(* PLC project Thermostats, Actility iec61131 1.0.231, author Laurent Nicq *)
(* stored: creationDateTime 2013-04-23T20:30:50, version V1.0.0, modificationDateTime 2013-07-22T15:08:27 *)

FUNCTION_BLOCK Heating_TH_PWM
  VAR_INPUT
    PWM2_Start : BOOL;
    PWM2_Period : TIME;
  END_VAR
  VAR
    PWM2_Running_ON_Time : TIME;
    PWM2_Ratio : DINT;
    PWM2_Limit_Low : DINT := 0;
  END_VAR
  VAR_INPUT
    PWM2_Limit_High : DINT;  (* If not set as INPUT, put 100.0 as initial value *)
  END_VAR
  VAR
    PWM_Ratio_Factor : DINT := 100;
    PWM2_ResetMode : DINT := 0;  (* For simulation *)
    PWM_Time_ON : TIME;
  END_VAR
  VAR_OUTPUT
    PWM2_Out : BOOL;
  END_VAR
  VAR_INPUT
    Setpoint : REAL;
    Temperature_Inside : REAL;
    Proportional_Inside : REAL;
    Temperature_Outside : REAL;
    Proportional_Outside : REAL;
  END_VAR
  VAR
    Inside_Demand : REAL;
    Outside_Demand : REAL;
    Demand_Factor : REAL := 100.0;
    PWM_HEATING : PWM_GENERATOR;
  END_VAR
  VAR  (* added by the conversion: wires and edge detectors of the diagram *)
    _SUB32_OUT : REAL;
    _MUL31_OUT : REAL;
    _SUB2_OUT : REAL;
    _MUL1_OUT : REAL;
    _ADD37_OUT : REAL;
    _MUL38_OUT : REAL;
    _REAL_TO_DINT41_OUT : DINT;
  END_VAR

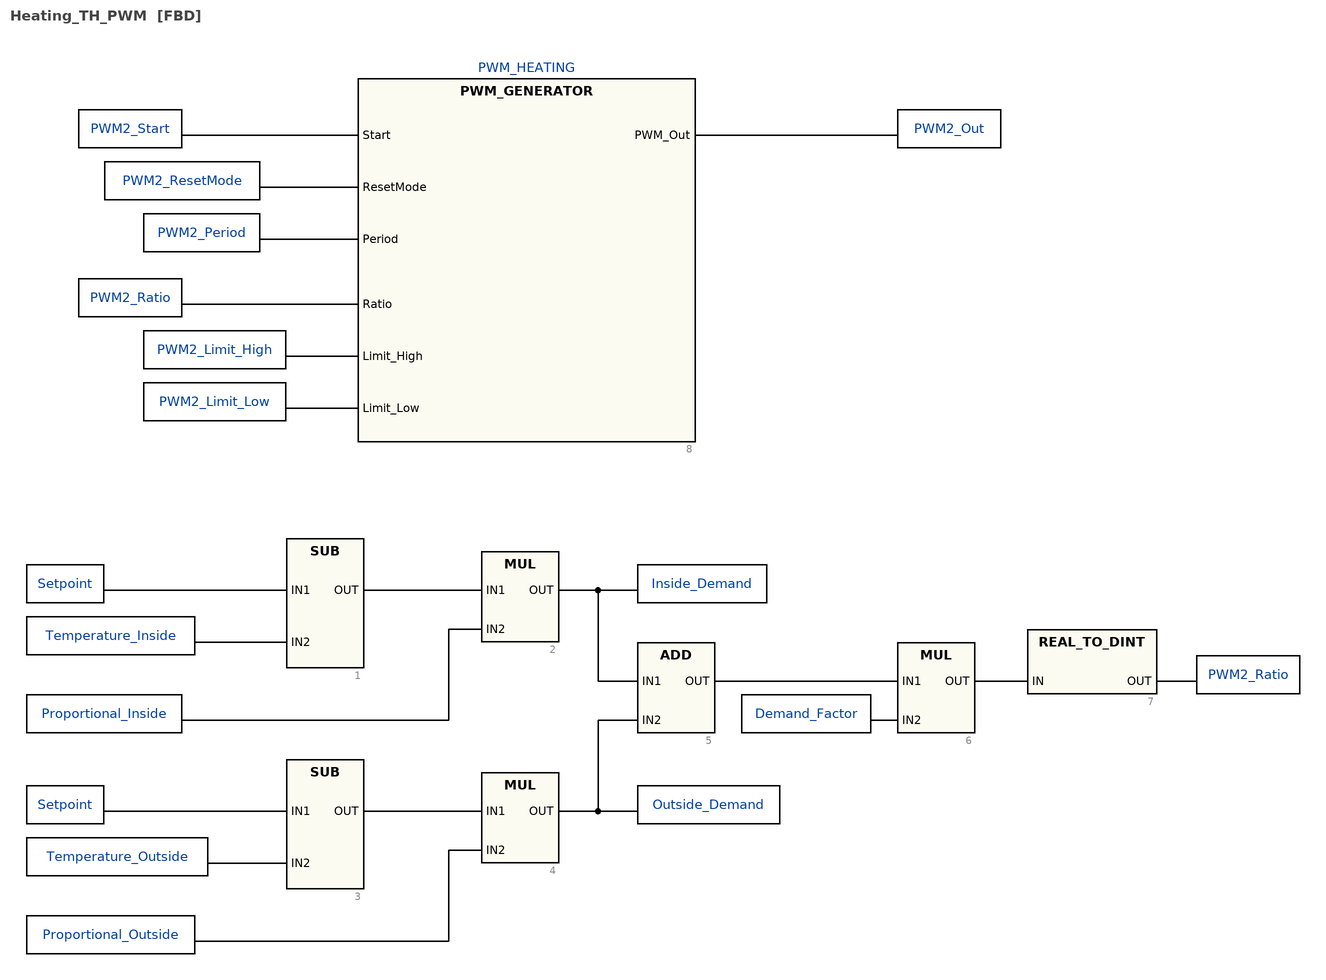
(* FBD diagram, written out as Structured Text *)
_SUB32_OUT := Setpoint - Temperature_Inside;
_MUL31_OUT := _SUB32_OUT * Proportional_Inside;
_SUB2_OUT := Setpoint - Temperature_Outside;
_MUL1_OUT := _SUB2_OUT * Proportional_Outside;
_ADD37_OUT := _MUL31_OUT + _MUL1_OUT;
_MUL38_OUT := _ADD37_OUT * Demand_Factor;
_REAL_TO_DINT41_OUT := REAL_TO_DINT(_MUL38_OUT);
PWM_HEATING(Start := PWM2_Start, ResetMode := PWM2_ResetMode, Period := PWM2_Period, Ratio := PWM2_Ratio, Limit_High := PWM2_Limit_High, Limit_Low := PWM2_Limit_Low);
PWM2_Out := PWM_HEATING.PWM_Out;
Inside_Demand := _MUL31_OUT;
PWM2_Ratio := _REAL_TO_DINT41_OUT;
Outside_Demand := _MUL1_OUT;
END_FUNCTION_BLOCK

PROGRAM Thermostat_PWM_DINT
  VAR
    TH_Period : TIME := T#20s;  (* Period in Second *)
    TH_PWM_Start : BOOL := FALSE;  (* Needs RISING Edge to start *)
    TH_Ratio_Limit_High : DINT := 100;  (* Ratio Limit High in % *)
    TH_Setpoint : REAL := 28.0;
  END_VAR
  VAR_EXTERNAL
    TH_Temp_Inside : REAL;
  END_VAR
  VAR
    TH_Temp_Outside : REAL := 12.0;
    TH_PROP_Inside : REAL := 0.5;
    TH_PROP_Outside : REAL := 0.0;
  END_VAR
  VAR_EXTERNAL
    TH_Output : BOOL;  (* PWM result *)
  END_VAR
  VAR
    Heating_Thermostat_1 : Heating_TH_PWM;
  END_VAR
  VAR  (* added by the conversion: wires and edge detectors of the diagram *)
    _NOT13_OUT : BOOL;
  END_VAR

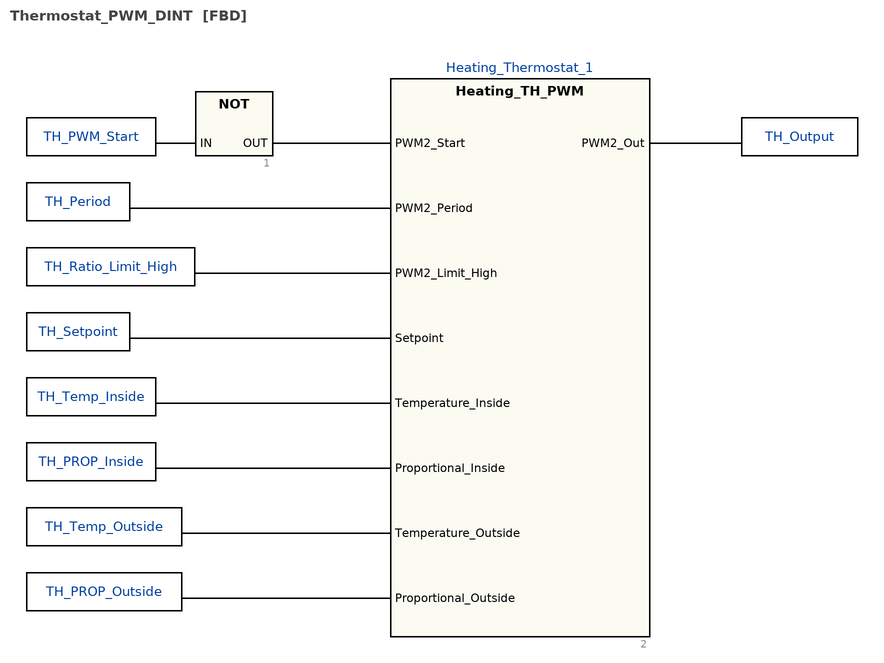
(* FBD diagram, written out as Structured Text *)
_NOT13_OUT := NOT TH_PWM_Start;
Heating_Thermostat_1(PWM2_Start := _NOT13_OUT, PWM2_Period := TH_Period, PWM2_Limit_High := TH_Ratio_Limit_High, Setpoint := TH_Setpoint, Temperature_Inside := TH_Temp_Inside, Proportional_Inside := TH_PROP_Inside, Temperature_Outside := TH_Temp_Outside, Proportional_Outside := TH_PROP_Outside);
TH_Output := Heating_Thermostat_1.PWM2_Out;
END_PROGRAM

CONFIGURATION config
  RESOURCE Thermostat1 ON PLC
    VAR_GLOBAL
      TH_Temp_Inside AT %IX1.1 : REAL;
      TH_Output AT %OX2.1 : BOOL;
    END_VAR
    TASK task1(INTERVAL := T#250ms, PRIORITY := 0);
    PROGRAM PWM1 WITH task1 : Thermostat_PWM_DINT;
  END_RESOURCE
END_CONFIGURATION
